// Mitsubishi GX Works2 project: Project_final2   PLC: Q01U

PROGRAM Conveyor
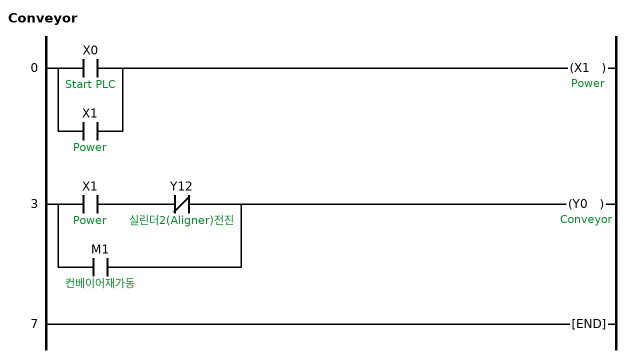
0     LD      X0  ; Start PLC
      OR      X1  ; Power
      OUT     X1  ; Power
3     LD      X1  ; Power
      ANI     Y12  ; 실린더2(Aligner)전진
      OR      M1  ; 컨베이어재가동
      OUT     Y0  ; Conveyor
7     END
END_PROGRAM

PROGRAM BoxAlign
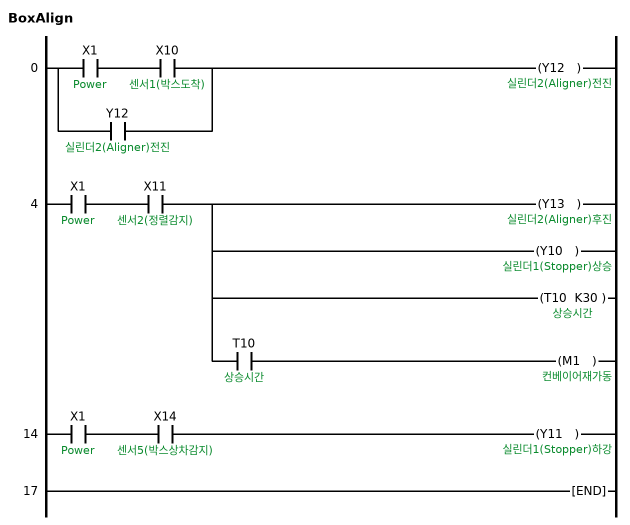
0     LD      X1  ; Power
      AND     X10  ; 센서1(박스도착)
      OR      Y12  ; 실린더2(Aligner)전진
      OUT     Y12  ; 실린더2(Aligner)전진
4     LD      X1  ; Power
      AND     X11  ; 센서2(정렬감지)
      OUT     Y13  ; 실린더2(Aligner)후진
      OUT     Y10  ; 실린더1(Stopper)상승
      OUT     T10 K30  ; 상승시간
      AND     T10  ; 상승시간
      OUT     M1  ; 컨베이어재가동
14    LD      X1  ; Power
      AND     X14  ; 센서5(박스상차감지)
      OUT     Y11  ; 실린더1(Stopper)하강
17    END
END_PROGRAM

PROGRAM BoxSort
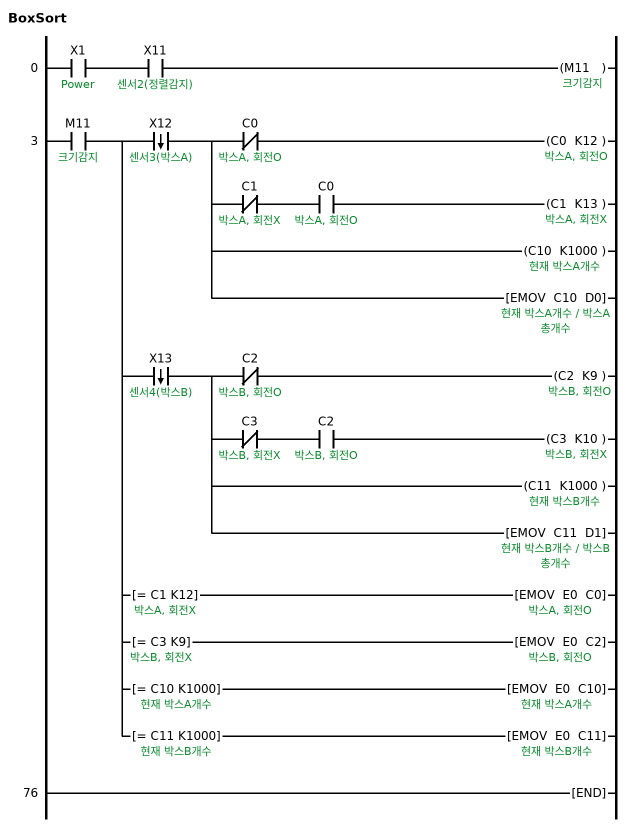
0     LD      X1  ; Power
      AND     X11  ; 센서2(정렬감지)
      OUT     M11  ; 크기감지
3     LD      M11  ; 크기감지
      MPS
      ANDF    X12  ; 센서3(박스A)
      MPS
      ANI     C0  ; 박스A, 회전O
      OUT     C0 K12  ; 박스A, 회전O
      MRD
      ANI     C1  ; 박스A, 회전X
      AND     C0  ; 박스A, 회전O
      OUT     C1 K13  ; 박스A, 회전X
      MPP
      OUT     C10 K1000  ; 현재 박스A개수
      EMOV    C10 D0  ; 박스A 총개수
      MRD
      ANDF    X13  ; 센서4(박스B)
      MPS
      ANI     C2  ; 박스B, 회전O
      OUT     C2 K9  ; 박스B, 회전O
      MRD
      ANI     C3  ; 박스B, 회전X
      AND     C2  ; 박스B, 회전O
      OUT     C3 K10  ; 박스B, 회전X
      MPP
      OUT     C11 K1000  ; 현재 박스B개수
      EMOV    C11 D1  ; 박스B 총개수
      MRD
      AND=    C1 K12  ; 박스A, 회전X
      EMOV    E0 C0
      MRD
      AND=    C3 K9  ; 박스B, 회전X
      EMOV    E0 C2
      MRD
      AND=    C10 K1000  ; 현재 박스A개수
      EMOV    E0 C10
      MPP
      AND=    C11 K1000  ; 현재 박스B개수
      EMOV    E0 C11
76    END
END_PROGRAM

PROGRAM BoxMove
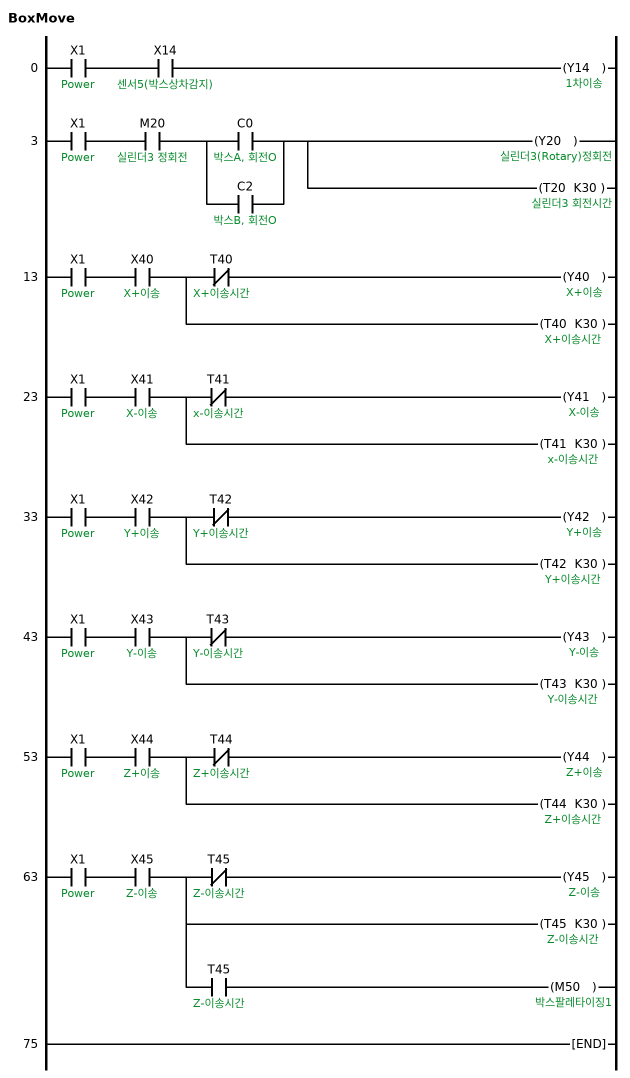
0     LD      X1  ; Power
      AND     X14  ; 센서5(박스상차감지)
      OUT     Y14  ; 1차이송
3     LD      X1  ; Power
      AND     M20  ; 실린더3 정회전
      LD      C0  ; 박스A, 회전O
      OR      C2  ; 박스B, 회전O
      ANB
      OUT     Y20  ; 실린더3(Rotary)정회전
      OUT     T20 K30  ; 실린더3 회전시간
13    LD      X1  ; Power
      AND     X40  ; X+이송
      MPS
      ANI     T40  ; X+이송시간
      OUT     Y40  ; X+이송
      MPP
      OUT     T40 K30  ; X+이송시간
23    LD      X1  ; Power
      AND     X41  ; X-이송
      MPS
      ANI     T41  ; x-이송시간
      OUT     Y41  ; X-이송
      MPP
      OUT     T41 K30  ; x-이송시간
33    LD      X1  ; Power
      AND     X42  ; Y+이송
      MPS
      ANI     T42  ; Y+이송시간
      OUT     Y42  ; Y+이송
      MPP
      OUT     T42 K30  ; Y+이송시간
43    LD      X1  ; Power
      AND     X43  ; Y-이송
      MPS
      ANI     T43  ; Y-이송시간
      OUT     Y43  ; Y-이송
      MPP
      OUT     T43 K30  ; Y-이송시간
53    LD      X1  ; Power
      AND     X44  ; Z+이송
      MPS
      ANI     T44  ; Z+이송시간
      OUT     Y44  ; Z+이송
      MPP
      OUT     T44 K30  ; Z+이송시간
63    LD      X1  ; Power
      AND     X45  ; Z-이송
      MPS
      ANI     T45  ; Z-이송시간
      OUT     Y45  ; Z-이송
      MPP
      OUT     T45 K30  ; Z-이송시간
      AND     T45  ; Z-이송시간
      OUT     M50  ; 박스팔레타이징1
75    END
END_PROGRAM

PROGRAM Pallet
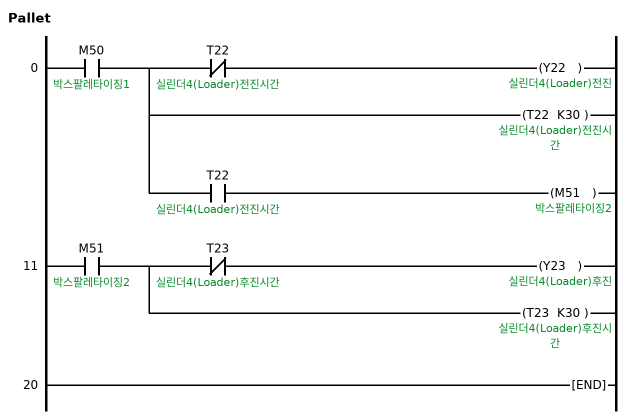
0     LD      M50  ; 박스팔레타이징1
      MPS
      ANI     T22  ; 실린더4(Loader)전진시간
      OUT     Y22  ; 실린더4(Loader)전진
      MPP
      OUT     T22 K30  ; 실린더4(Loader)전진시간
      AND     T22  ; 실린더4(Loader)전진시간
      OUT     M51  ; 박스팔레타이징2
11    LD      M51  ; 박스팔레타이징2
      MPS
      ANI     T23  ; 실린더4(Loader)후진시간
      OUT     Y23  ; 실린더4(Loader)후진
      MPP
      OUT     T23 K30  ; 실린더4(Loader)후진시간
20    END
END_PROGRAM

PROGRAM Change
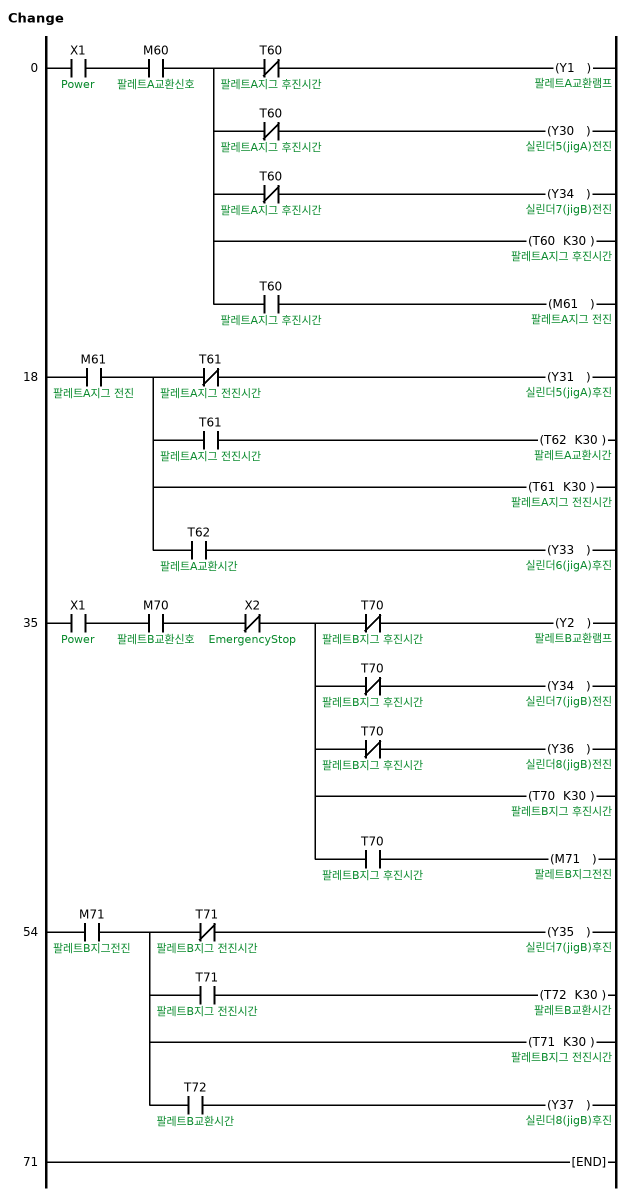
0     LD      X1  ; Power
      AND     M60  ; 팔레트A교환신호
      MPS
      ANI     T60  ; 팔레트A지그 후진시간
      OUT     Y1  ; 팔레트A교환램프
      MRD
      ANI     T60  ; 팔레트A지그 후진시간
      OUT     Y30  ; 실린더5(jigA)전진
      MRD
      ANI     T60  ; 팔레트A지그 후진시간
      OUT     Y34  ; 실린더7(jigB)전진
      MPP
      OUT     T60 K30  ; 팔레트A지그 후진시간
      AND     T60  ; 팔레트A지그 후진시간
      OUT     M61  ; 팔레트A지그 전진
18    LD      M61  ; 팔레트A지그 전진
      MPS
      ANI     T61  ; 팔레트A지그 전진시간
      OUT     Y31  ; 실린더5(jigA)후진
      MRD
      AND     T61  ; 팔레트A지그 전진시간
      OUT     T62 K30  ; 팔레트A교환시간
      MPP
      OUT     T61 K30  ; 팔레트A지그 전진시간
      AND     T62  ; 팔레트A교환시간
      OUT     Y33  ; 실린더6(jigA)후진
35    LD      X1  ; Power
      AND     M70  ; 팔레트B교환신호
      ANI     X2  ; EmergencyStop
      MPS
      ANI     T70  ; 팔레트B지그 후진시간
      OUT     Y2  ; 팔레트B교환램프
      MRD
      ANI     T70  ; 팔레트B지그 후진시간
      OUT     Y34  ; 실린더7(jigB)전진
      MRD
      ANI     T70  ; 팔레트B지그 후진시간
      OUT     Y36  ; 실린더8(jigB)전진
      MPP
      OUT     T70 K30  ; 팔레트B지그 후진시간
      AND     T70  ; 팔레트B지그 후진시간
      OUT     M71  ; 팔레트B지그전진
54    LD      M71  ; 팔레트B지그전진
      MPS
      ANI     T71  ; 팔레트B지그 전진시간
      OUT     Y35  ; 실린더7(jigB)후진
      MRD
      AND     T71  ; 팔레트B지그 전진시간
      OUT     T72 K30  ; 팔레트B교환시간
      MPP
      OUT     T71 K30  ; 팔레트B지그 전진시간
      AND     T72  ; 팔레트B교환시간
      OUT     Y37  ; 실린더8(jigB)후진
71    END
END_PROGRAM

// device comments not shown above
Y32  ; 실린더6(jigA)전진
Y50  ; 박스하차
Y60  ; 램프
M30  ; 박스 이송
M40  ; X+이송
M41  ; X-이송
M42  ; Y+이송
M43  ; Y-이송
M44  ; Z+이송
M45  ; Z-이송
M62  ; 팔레트B교환신호
T11  ; 실린더1후진시간
T50  ; 실린더4(Loader)작동시간
